// TIA Portal V21 export
DATA_BLOCK "DB_MES"   // DB1000
VERSION : 0.0
// stored: AutoNumber false, InstanceOfName AUX MES, InstanceOfType FB
"AUX MES"
   // VAR RETAIN
   //    DATI { S7_SetPoint := 'True'} : "UDT_MES";
   //    TOUT { S7_SetPoint := 'True'} : IEC_TIMER;
   //    FP1 : Bool := FALSE;
   //    FP2 : Bool := TRUE;
   //    COMM_ERROR : Bool := TRUE;
   //    IndexPID : Int := 8;
   //    AllarmePresenteSterilizzatore { ExternalVisible := 'False'; ExternalWritable := 'False'} : Bool := TRUE;
   //    AllarmePresentePID : Bool := FALSE;
   // END_VAR
BEGIN
   DATI.aux_to._0_0 := FALSE;
   DATI.aux_to._0_1 := FALSE;
   DATI.aux_to._0_2 := FALSE;
   DATI.aux_to._0_3 := FALSE;
   DATI.aux_to._0_4 := FALSE;
   DATI.aux_to._0_5 := FALSE;
   DATI.aux_to._0_6 := FALSE;
   DATI.aux_to._0_7 := FALSE;
   DATI.aux_to._1_0 := FALSE;
   DATI.aux_to._1_1 := TRUE;
   DATI.aux_to._1_2 := FALSE;
   DATI.aux_to._1_3 := FALSE;
   DATI.aux_to._1_4 := FALSE;
   DATI.aux_to._1_5 := FALSE;
   DATI.aux_to._1_6 := FALSE;
   DATI.aux_to._1_7 := FALSE;
   DATI."to"._bit._0_0 := FALSE;
   DATI."to"._bit._0_1 := FALSE;
   DATI."to"._bit._0_2 := FALSE;
   DATI."to"._bit._0_3 := FALSE;
   DATI."to"._bit._0_4 := TRUE;
   DATI."to"._bit._0_5 := FALSE;   // Funzionamento Pompa Mono/Pistoni
   DATI."to"._bit._0_6 := FALSE;
   DATI."to"._bit._0_7 := FALSE;
   DATI."to"._bit._1_0 := FALSE;
   DATI."to"._bit._1_1 := FALSE;
   DATI."to"._bit._1_2 := FALSE;
   DATI."to"._bit._1_3 := FALSE;
   DATI."to"._bit._1_4 := FALSE;
   DATI."to"._bit._1_5 := FALSE;
   DATI."to"._bit._1_6 := FALSE;
   DATI."to"._bit._1_7 := FALSE;
   DATI."to"._bit._2_0 := FALSE;
   DATI."to"._bit._2_1 := FALSE;
   DATI."to"._bit._2_2 := FALSE;
   DATI."to"._bit._2_3 := FALSE;
   DATI."to"._bit._2_4 := FALSE;
   DATI."to"._bit._2_5 := FALSE;
   DATI."to"._bit._2_6 := FALSE;
   DATI."to"._bit._2_7 := FALSE;
   DATI."to"._bit._3_0 := FALSE;
   DATI."to"._bit._3_1 := FALSE;
   DATI."to"._bit._3_2 := FALSE;
   DATI."to"._bit._3_3 := FALSE;
   DATI."to"._bit._3_4 := FALSE;
   DATI."to"._bit._3_5 := FALSE;
   DATI."to"._bit._3_6 := FALSE;
   DATI."to"._bit._3_7 := FALSE;
   DATI."to"._dint._0_00 := 1;
   DATI."to"._dint._0_01 := 0;
   DATI."to"._dint._0_02 := 0;
   DATI."to"._dint._0_03 := 0;
   DATI."to"._dint._0_04 := 62.80744;
   DATI."to"._dint._0_05 := 41.04094;
   DATI."to"._dint._0_06 := 69.92146;
   DATI."to"._dint._0_07 := 58.15972;
   DATI."to"._dint._0_08 := 0.0;
   DATI."to"._dint._0_09 := 116.0;
   DATI."to"._dint._0_010 := 109.4016;
   DATI."to"._dint._0_011 := 35.8;
   DATI."to"._dint._0_012 := 5505.907;
   DATI."to"._dint._0_013 := 0.1989294;
   DATI."to"._dint._0_014 := 0.0;
   DATI."to"._dint._0_015 := 0.0;
   DATI."to"._dint._0_016 := 0.0;
   DATI."to"._dint._0_017 := 3.255208;
   DATI."to"._dint._0_018 := 0.0;
   DATI."to"._dint._0_019 := 0.0;
   DATI."to"._dint._0_020 := 0.0;
   DATI."to"._dint._0_021 := 0.0;
   DATI."to"._dint._0_022 := 0.0;
   DATI."to"._dint._0_023 := 16.27604;
   DATI."to"._dint._0_024 := 13.02083;
   DATI."to"._dint._0_025 := 13.02083;
   DATI."to"._dint._0_026 := 0.0;
   DATI."to"._dint._0_027 := 7.595486;
   DATI."to"._dint._0_028 := 9.765625;
   DATI."to"._dint._0_029 := 7.595486;
   DATI."to"._dint._0_030 := 2.170139;
   DATI."to"._dint._0_031 := 2.170139;
   DATI."to"._dint._0_032 := 0.0;
   DATI."to"._dint._0_033 := 23.7;
   DATI."to"._dint._0_034 := 24.0;
   DATI."to"._dint._0_035 := 23.0;
   DATI."to"._string._0_00 := 'passata';
   DATI."to"._string._0_01 := '';
   DATI."to"._string._0_02 := '';
   DATI."to"._string._0_03 := '';
   DATI."to"._string._0_04 := '';
   DATI."to"._string._0_05 := '';
   DATI."to"._string._0_06 := '';
   DATI._aux_from._0_0 := FALSE;
   DATI._aux_from._0_1 := FALSE;
   DATI._aux_from._0_2 := FALSE;
   DATI._aux_from._0_3 := FALSE;
   DATI._aux_from._0_4 := FALSE;
   DATI._aux_from._0_5 := FALSE;
   DATI._aux_from._0_6 := FALSE;
   DATI._aux_from._0_7 := FALSE;
   DATI._aux_from._1_0 := FALSE;
   DATI._aux_from._1_1 := FALSE;
   DATI._aux_from._1_2 := FALSE;
   DATI._aux_from._1_3 := FALSE;
   DATI._aux_from._1_4 := FALSE;
   DATI._aux_from._1_5 := FALSE;
   DATI._aux_from._1_6 := FALSE;
   DATI._aux_from._1_7 := FALSE;
   DATI.from._bit._0_0 := FALSE;
   DATI.from._bit._0_1 := FALSE;
   DATI.from._bit._0_2 := FALSE;
   DATI.from._bit._0_3 := FALSE;
   DATI.from._bit._0_4 := FALSE;
   DATI.from._bit._0_5 := FALSE;
   DATI.from._bit._0_6 := FALSE;
   DATI.from._bit._0_7 := FALSE;
   DATI.from._bit._1_0 := FALSE;
   DATI.from._bit._1_1 := FALSE;
   DATI.from._bit._1_2 := FALSE;
   DATI.from._bit._1_3 := FALSE;
   DATI.from._bit._1_4 := FALSE;
   DATI.from._bit._1_5 := FALSE;
   DATI.from._bit._1_6 := FALSE;
   DATI.from._bit._1_7 := FALSE;
   DATI.from._bit._2_0 := FALSE;
   DATI.from._bit._2_1 := FALSE;
   DATI.from._bit._2_2 := FALSE;
   DATI.from._bit._2_3 := FALSE;
   DATI.from._bit._2_4 := FALSE;
   DATI.from._bit._2_5 := FALSE;
   DATI.from._bit._2_6 := FALSE;
   DATI.from._bit._2_7 := FALSE;
   DATI.from._bit._3_0 := FALSE;
   DATI.from._bit._3_1 := FALSE;
   DATI.from._bit._3_2 := FALSE;
   DATI.from._bit._3_3 := FALSE;
   DATI.from._bit._3_4 := FALSE;
   DATI.from._bit._3_5 := FALSE;
   DATI.from._bit._3_6 := FALSE;
   DATI.from._bit._3_7 := FALSE;
   DATI.from._dint._0_00 := 1_987_051_520;
   DATI.from._dint._0_01 := 0;
   DATI.from._dint._0_02 := 0;
   DATI.from._dint._0_03 := 0;
   DATI.from._dint._0_04 := 0;
   DATI.from._dint._0_05 := 0;
   DATI.from._dint._0_06 := 0;
   DATI.from._dint._0_07 := 0;
   DATI.from._dint._0_08 := 0;
   DATI.from._dint._0_09 := 0;
   DATI.from._dint._0_010 := 0;
   DATI.from._dint._0_011 := 0;
   DATI.from._dint._0_012 := 0;
   DATI.from._dint._0_013 := 0;
   DATI.from._dint._0_014 := 0;
   DATI.from._dint._0_015 := 0;
   DATI.from._dint._0_016 := 0;
   DATI.from._dint._0_017 := 0;
   DATI.from._dint._0_018 := 0;
   DATI.from._dint._0_019 := 0;
   DATI.from._dint._0_020 := 0;
   DATI.from._dint._0_021 := 0;
   DATI.from._dint._0_022 := 0;
   DATI.from._dint._0_023 := 0;
   DATI.from._dint._0_024 := 0;
   DATI.from._dint._0_025 := 0;
   DATI.from._dint._0_026 := 0;
   DATI.from._dint._0_027 := 0;
   DATI.from._dint._0_028 := 0;
   DATI.from._dint._0_029 := 0;
   DATI.from._dint._0_030 := 0;
   DATI.from._dint._0_031 := 0;
   DATI.from._dint._0_032 := 0;
   DATI.from._dint._0_033 := 0;
   DATI.from._dint._0_034 := 0;
   DATI.from._dint._0_035 := 0;
   DATI.from._string._0_00 := 'Rototermo Goglio';
   DATI.from._string._0_01 := '';
   DATI.from._string._0_02 := '';
   DATI.from._string._0_03 := '';
   DATI.from._string._0_04 := '';
   DATI.from._string._0_05 := '';
   DATI.from._string._0_06 := '';
   TOUT.PT := T#5S;
   TOUT.IN := TRUE;
END_DATA_BLOCK
